// SIMATIC S7-200 project (STEP 7-Micro/WIN), CPU 224 CN REL 02.01

SYMBOL_TABLE 用户定义1
PN_3             VD521    // 3段脉冲数
T_INCR_3         VW519    // 3段周期增量
T_3              VW517    // 3段初始周期
PN_2             VD513    // 2段脉冲数
T_INCR_2         VW511    // 2段周期增量
T_2              VW509    // 2段初始周期
PN_1             VD505    // 1段脉冲数
T_INCR_1         VW503    // 1段周期增量
T_1              VW501    // 1段初始周期
END_SYMBOL_TABLE

ORGANIZATION_BLOCK 主程序:OB1
TITLE=程序通过监控启动信号、方向控制信号、速度控制信号和使能信号，直接控制步进电机的运行参数。
// 启动信号控制电机运行状态，当启动信号为真时电机启动，否则停止；
// 方向控制信号控制电机方向，当方向控制信号为真时电机正转，否则反转；
// 速度控制信号控制电机速度，当速度控制信号为真时电机高速运行，否则低速运行；
// 使能信号控制电机使能，当使能信号为真时电机启用，否则禁用；
// 当需要将工件移动到指定位置时，可以通过HMI按钮触发脉冲发生器，程序会调用脉冲发生器子程序，通过设置相关参数并调用PLS指令，生成脉冲信号，控制步进电机移动到指定位置。
BEGIN
Network 1 // 网络标题
// 网络注释
LD     V0.0
=      Q2.5
Network 2
LD     V0.1
=      Q2.0
Network 3
LD     V0.2
=      Q1.1
Network 4
LD     V0.3
=      Q0.2
Network 5
LD     V0.4
EU
CALL   SBR_0:SBR0
END_ORGANIZATION_BLOCK

SUBROUTINE_BLOCK SBR_0:SBR0
TITLE=子程序注释
BEGIN
Network 1 // 网络标题
// 多段，微秒
LD     SM0.0
MOVB   16#A0, SMB67
Network 2
// 起始偏移地址
LD     SM0.0
MOVW   500, SMW168
Network 3
LD     SM0.0
PLS    0
END_SUBROUTINE_BLOCK

DATA_BLOCK_TAB 用户定义1
BEGIN
//数据页注释
//按 F1 键获取帮助和示范数据页
VB500    3                   //总段数
         T_1                 //初始周期
         T_INCR_1            //周期增量
         PN_1                //脉冲数
         T_2                 //初始周期
         T_INCR_2, 0         //周期增量
         PN_2                //脉冲数
         T_3                 //初始周期
         T_INCR_3            //周期增量
         PN_3                //脉冲数
END_DATA_BLOCK_TAB
